{attribute 'GeneratedUsingTerminal: EL2034-0000-0018'}
{attribute addProperty BoxType "EL2034-0000-0018"}
{attribute addProperty Id "EtcSlaveTerminalBaseDiag_1AT %I*Diag_A72B1E171Diag_2AT %I*Diag_A72B1E171Diag_3AT %I*Diag_A72B1E171Diag_4AT %I*Diag_A72B1E171Channel_1AT %Q*Channel_42CA91F71Channel_2AT %Q*Channel_42CA91F71Channel_3AT %Q*Channel_42CA91F71Channel_4AT %Q*Channel_42CA91F71WcStateAT %I*WcState_9091E0EB2InfoDataAT %I*InfoData_6F19DB2B2"}
{attribute addProperty CRC "1999745160"}
{attribute addProperty Size "12"}
TYPE EL2034_7731B088 EXTENDS EtcSlaveTerminalBase :
STRUCT
	{attribute addProperty Name "Diag_1"}
	Diag_1 : Diag_A72B1E17;
	{attribute addProperty Name "Diag_2"}
	Diag_2 : Diag_A72B1E17;
	{attribute addProperty Name "Diag_3"}
	Diag_3 : Diag_A72B1E17;
	{attribute addProperty Name "Diag_4"}
	Diag_4 : Diag_A72B1E17;
	{attribute addProperty Name "Channel_1"}
	Channel_1 : Channel_42CA91F7;
	{attribute addProperty Name "Channel_2"}
	Channel_2 : Channel_42CA91F7;
	{attribute addProperty Name "Channel_3"}
	Channel_3 : Channel_42CA91F7;
	{attribute addProperty Name "Channel_4"}
	Channel_4 : Channel_42CA91F7;
	{attribute addProperty Name "WcState"}
	WcState : WcState_9091E0EB;
	{attribute addProperty Name "InfoData"}
	InfoData : InfoData_6F19DB2B;
END_STRUCT
END_TYPE

(* stored: Version 1.2.0.0, ProductVersion 3.1.4024.9
   DUT EL2034_7731B088: Id {540e704e-0ebf-4bc5-be1d-1e0936d0ff71} *)
